TYPE "SpeedMachine_DataIn"
VERSION : 0.1
// Block: SpeedMachine_DataIn
   STRUCT
      PB : Ax_PB;
      Fan_M_ThermalProtection : Bool;
      Fan_M_Feedback : Bool;
      Brake_M_Q : Bool;
      Brake_M_Feedback : Bool;
   END_STRUCT;

END_TYPE
